//{attribute 'qualified_only'}
//{attribute 'strict'}
{attribute 'to_string'}

TYPE E_RS_Cycles :
(
	Idle := 0,
	DeadAirEvac,
	SteamDesorption,
	VacCooling,
	AirRepress,
	Adsorption,
	Estop,
	SafeShutdown,
	Error := 9
);
END_TYPE

(* stored: Version 1.1.0.1, ProductVersion 3.1.4024.12
   DUT E_RS_Cycles: Id {385ae84b-766b-4002-b912-752d54a20d2d} *)
